FUNCTION_BLOCK FB_Robot_Mitsubishi_ReceivePacket
VAR_INPUT
END_VAR
VAR_OUTPUT
	LastReceivedPacket				: STRING(255);
	LastReceivedPacketID			: DINT;
END_VAR
VAR_IN_OUT
	ConnectionRef					: FB_ClientServerConnection;											//
END_VAR
VAR
	fbReceive						: FB_SocketReceive;														// Receive data trough TCP IP.
	aInputBuffer					: ARRAY[0..255] OF BYTE;												// 
	bBusy							: BOOL;
END_VAR

IF ConnectionRef.eState = eSOCKET_CONNECTED AND (NOT ConnectionRef.bBusy) THEN
	IF NOT bBusy THEN
		fbReceive( bExecute := FALSE);	
		fbReceive( 	sSrvNetId	:= ConnectionRef.sSrvNetID,
					hSocket		:= ConnectionRef.hSocket,
					cbLen		:= SIZEOF(aInputBuffer),
					pDest		:= ADR(aInputBuffer),
					tTimeout	:= T#100MS,
					bExecute	:= TRUE);
		bBusy := TRUE;
	ELSE
		fbReceive( bExecute := FALSE);
		IF (NOT fbReceive.bBusy) THEN
			bBusy := FALSE;
			IF fbReceive.nRecBytes > 10 THEN															// 8 Bytes for packet ID and 2 bytes for <LF><CR>
				LastReceivedPacketID := 0;
				LastReceivedPacket := '';
				MEMCPY(ADR(LastReceivedPacket),														// Copy the packet header data.
					ADR(aInputBuffer),																// Could trim the <LF><CR> flags.
					fbReceive.nRecBytes);
				FB_HEXSTR_TO_DINT(in := LEFT(LastReceivedPacket, 8),
					out => LastReceivedPacketID);
				MEMSET(ADR(aInputBuffer),
					0,
					SIZEOF(aInputBuffer));
			ELSE
				MEMSET(ADR(aInputBuffer),
					0,
					SIZEOF(aInputBuffer));
			END_IF
		END_IF
	END_IF
ELSE
	fbReceive( bExecute := FALSE );
END_IF

END_FUNCTION_BLOCK

(* stored: Version 1.1.0.1, ProductVersion 3.1.4024.2
   POU FB_Robot_Mitsubishi_ReceivePacket: Id {52dc5b5e-1f9d-410f-9612-1286f69acc03}, SpecialFunc None *)
